FUNCTION_BLOCK E_TRAIN (* Generation of a finite train of events *)
  (* Standard: 61499-2 *)
  (* Version 0.3, 2008-06-03, JHC, Holobloc Inc, Added package declaration. *)
  (* Version 0.2, 2004-04-18, JHC, Rockwell Automation, Updated documentation. *)
  (* Version 0.1, 2002-01-30, JHC, Rockwell Automation, XML (SIFB) version *)
  (* Version 0.0, 1998-09-11, JHC, Rockwell Automation, SRC (composite) version *)
  (* Compiler header: package fb.rt.events; *)
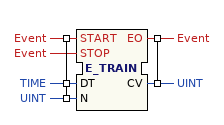
  EVENT_INPUT
    START WITH DT, N;
    STOP;
  END_EVENT
  EVENT_OUTPUT
    EO WITH CV; (* N events at period DT,starting at DT after START *)
  END_EVENT
  VAR_INPUT
    DT : TIME; (* Period between events *)
    N : UINT; (* Number of events to generate *)
  END_VAR
  VAR_OUTPUT
    CV : UINT; (* EO index(0 N-1) *)
  END_VAR
  SERVICE E_TRAIN/resource
    SEQUENCE normal_operation (* N=3 *)
      E_TRAIN.START(DT);
      -> E_TRAIN.EO(CV=0);
      -> E_TRAIN.EO(CV=1);
      -> E_TRAIN.EO(CV=2);
    END_SEQUENCE
    SEQUENCE no_restart (* N=3 *)
      E_TRAIN.START(DT);
      -> E_TRAIN.EO(CV=0);
      E_TRAIN.START(DT);
      -> E_TRAIN.EO(CV=1);
      -> E_TRAIN.EO(CV=2);
    END_SEQUENCE
    SEQUENCE cycle_canceled
      E_TRAIN.START(DT);
      -> E_TRAIN.EO(CV=0);
      E_TRAIN.STOP();
    END_SEQUENCE
  END_SERVICE
END_FUNCTION_BLOCK
